{attribute 'Tc2GvlVarNames'}
VAR_GLOBAL
(*Master*)
(*Gerät 4 (CX5130-0121-M310), BOX 01*)
(*DP/DP-Kopppler*)
(*DP_State*)
(*
	R1_B01_PB_Zustand						AT %I*: USINT;
(*Daten*)
	R1_B01_StatusModule_I_Byte_1			AT %I*: USINT;
	R1_B01_StatusModule_I_Byte_2			AT %I*: USINT;
	R1_B01_StatusModule_I_Byte_5			AT %I*: USINT;
	R1_B01_StatusModule_I_Byte_6			AT %I*: USINT;
	R1_B01_ControlModule_O					AT %Q* :ARRAY [0..4] OF USINT;
	R1_B01_VolumeFlow_I						AT %I* :UDINT;
	R1_B01_PumpLiquidTemp_I					AT %I* :UDINT;
	R1_B01_OperationTime_I					AT %I* :UDINT;
	R1_B01_ActualSetpoint_I					AT %I* :UDINT;
	R1_B01_Frequency_I						AT %I* :UDINT;
	R1_B01_UserSetpoint_I					AT %I* :UDINT;
	R1_B01_DiffPressure_I					AT %I* :UDINT;
	R1_B01_RemoteTemp2						AT %I* :UDINT;
	R1_B01_HeatEnergyCounter_I				AT %I* :UDINT;
	R1_B01_HeatDiffTemp						AT %I* :UDINT;
	R1_B01_HeatPower						AT %I* :UDINT;  (* B0_SequenceNumber(1),B1AddressGenib(30),B2Class(11),B3Operation_Lenght(1),B4Data1(ID.34),Data(B5-B8) *)
	R1_B01_DirectDataReques_Temp_Geni		AT %Q* :PB_GenibusType;		(*ARRAY [0..8] OF USINT := 1, 255, 11, 1, 34, 0, 0, 0, 0;*)
	R1_B01_DirectDataReply_Temp_Geni		AT %I* :PB_GenibusType;		(*ARRAY [0..8] OF USINT;*)



	R1_B01_NumberOfStarts					AT %I*	: 	UDINT;
	R1_B01_ActualSetpoint					AT %I*	:	UDINT;
	R1_B01_OperationTime					AT %I*	: 	UDINT;
	R1_B01_Speed							AT %I*	:	UDINT;
	R1_B01_Energy							AT %I*	: 	UDINT;
	R1_B01_Power							AT %I*	:	UDINT;
	R1_B01_PowerElectronicsTemp				AT %I*	:	UDINT;
	R1_B01_FaultCode						AT %I*	:	USINT;
	R1_B01_Volume							AT %I*	:	UDINT;
	R1_B01_WarningCode						AT %I*	:	USINT;

(*Gerät 4 (CX5130-0121-M310), BOX 02*)
(*DP/DP-Kopppler*)
(*DP_State*)
	R1_B02_PB_Zustand						AT %I*: USINT;
(*Daten*)
	R1_B02_StatusModule_I_Byte_1			AT %I*: USINT;
	R1_B02_StatusModule_I_Byte_2			AT %I*: USINT;
	R1_B02_StatusModule_I_Byte_5			AT %I*: USINT;
	R1_B02_StatusModule_I_Byte_6			AT %I*: USINT;
	R1_B02_ControlModule_O					AT %Q* :ARRAY [0..4] OF USINT;
	R1_B02_VolumeFlow_I						AT %I* :UDINT;
	R1_B02_PumpLiquidTemp_I					AT %I* :UDINT;
	R1_B02_OperationTime_I					AT %I* :UDINT;
	R1_B02_ActualSetpoint_I					AT %I* :UDINT;
	R1_B02_Frequency_I						AT %I* :UDINT;
	R1_B02_UserSetpoint_I					AT %I* :UDINT;
	R1_B02_DiffPressure_I					AT %I* :UDINT;
	R1_B02_RemoteTemp2						AT %I* :UDINT;
	R1_B02_HeatEnergyCounter_I				AT %I* :UDINT;
	R1_B02_HeatDiffTemp						AT %I* :UDINT;
	R1_B02_HeatPower						AT %I* :UDINT;(* B0_SequenceNumber(1),B1AddressGenib(30),B2Class(11),B3Operation_Lenght(1),B4Data1(ID.34),Data(B5-B8) *)
	R1_B02_DirectDataReques_Temp_Geni		AT %Q* :PB_GenibusType;
	R1_B02_DirectDataReply_Temp_Geni		AT %I* :PB_GenibusType;


	R1_B02_NumberOfStarts					AT %I*	: 	UDINT;
	R1_B02_ActualSetpoint					AT %I*	:	UDINT;
	R1_B02_OperationTime					AT %I*	: 	UDINT;
	R1_B02_Speed							AT %I*	:	UDINT;
	R1_B02_Energy							AT %I*	: 	UDINT;
	R1_B02_Power							AT %I*	:	UDINT;
	R1_B02_PowerElectronicsTemp				AT %I*	:	UDINT;
	R1_B02_FaultCode						AT %I*	:	USINT;
	R1_B02_Volume							AT %I*	:	UDINT;
	R1_B02_WarningCode						AT %I*	:	USINT;

(*Gerät 4 (CX5130-0121-M310), BOX 03*)
(*DP/DP-Kopppler*)
(*DP_State*)
	R1_B03_PB_Zustand						AT %I*: USINT;
(*Daten*)
	R1_B03_StatusModule_I_Byte_1			AT %I*: USINT;
	R1_B03_StatusModule_I_Byte_2			AT %I*: USINT;
	R1_B03_StatusModule_I_Byte_5			AT %I*: USINT;
	R1_B03_StatusModule_I_Byte_6			AT %I*: USINT;
	R1_B03_ControlModule_O					AT %Q* :ARRAY [0..4] OF USINT;
	R1_B03_VolumeFlow_I						AT %I* :UDINT;
	R1_B03_PumpLiquidTemp_I					AT %I* :UDINT;
	R1_B03_OperationTime_I					AT %I* :UDINT;
	R1_B03_ActualSetpoint_I					AT %I* :UDINT;
	R1_B03_Frequency_I						AT %I* :UDINT;
	R1_B03_UserSetpoint_I					AT %I* :UDINT;
	R1_B03_DiffPressure_I					AT %I* :UDINT;
	R1_B03_RemoteTemp2						AT %I* :UDINT;
	R1_B03_HeatEnergyCounter_I				AT %I* :UDINT;
	R1_B03_HeatDiffTemp						AT %I* :UDINT;
	R1_B03_HeatPower						AT %I* :UDINT;(* B0_SequenceNumber(1),B1AddressGenib(30),B2Class(11),B3Operation_Lenght(1),B4Data1(ID.34),Data(B5-B8) *)
	R1_B03_DirectDataReques_Temp_Geni		AT %Q* :PB_GenibusType;
	R1_B03_DirectDataReply_Temp_Geni		AT %I* :PB_GenibusType;

	R1_B03_NumberOfStarts					AT %I*	: 	UDINT;
	R1_B03_ActualSetpoint					AT %I*	:	UDINT;
	R1_B03_OperationTime					AT %I*	: 	UDINT;
	R1_B03_Speed							AT %I*	:	UDINT;
	R1_B03_Energy							AT %I*	: 	UDINT;
	R1_B03_Power							AT %I*	:	UDINT;
	R1_B03_PowerElectronicsTemp				AT %I*	:	UDINT;
	R1_B03_FaultCode						AT %I*	:	USINT;
	R1_B03_Volume							AT %I*	:	UDINT;
	R1_B03_WarningCode						AT %I*	:	USINT;

(*Gerät 4 (CX5130-0121-M310), BOX 04*)
(*DP/DP-Kopppler*)
(*DP_State*)
	R1_B04_PB_Zustand						AT %I*: USINT;
(*Daten*)
	R1_B04_StatusModule_I_Byte_1			AT %I*: USINT;
	R1_B04_StatusModule_I_Byte_2			AT %I*: USINT;
	R1_B04_StatusModule_I_Byte_5			AT %I*: USINT;
	R1_B04_StatusModule_I_Byte_6			AT %I*: USINT;
	R1_B04_ControlModule_O					AT %Q* :ARRAY [0..4] OF USINT;
	R1_B04_VolumeFlow_I						AT %I* :UDINT;
	R1_B04_PumpLiquidTemp_I					AT %I* :UDINT;
	R1_B04_OperationTime_I					AT %I* :UDINT;
	R1_B04_ActualSetpoint_I					AT %I* :UDINT;
	R1_B04_Frequency_I						AT %I* :UDINT;
	R1_B04_UserSetpoint_I					AT %I* :UDINT;
	R1_B04_DiffPressure_I					AT %I* :UDINT;
	R1_B04_RemoteTemp2						AT %I* :UDINT;
	R1_B04_HeatEnergyCounter_I				AT %I* :UDINT;
	R1_B04_HeatDiffTemp						AT %I* :UDINT;
	R1_B04_HeatPower						AT %I* :UDINT;(* B0_SequenceNumber(1),B1AddressGenib(30),B2Class(11),B3Operation_Lenght(1),B4Data1(ID.34),Data(B5-B8) *)
	R1_B04_DirectDataReques_Temp_Geni		AT %Q* :PB_GenibusType;
	R1_B04_DirectDataReply_Temp_Geni		AT %I* :PB_GenibusType;


	R1_B04_NumberOfStarts					AT %I*	: 	UDINT;
	R1_B04_ActualSetpoint					AT %I*	:	UDINT;
	R1_B04_OperationTime					AT %I*	: 	UDINT;
	R1_B04_Speed							AT %I*	:	UDINT;
	R1_B04_Energy							AT %I*	: 	UDINT;
	R1_B04_Power							AT %I*	:	UDINT;
	R1_B04_PowerElectronicsTemp				AT %I*	:	UDINT;
	R1_B04_FaultCode						AT %I*	:	USINT;
	R1_B04_Volume							AT %I*	:	UDINT;
	R1_B04_WarningCode						AT %I*	:	USINT;


(*Gerät 4 (CX5130-0121-M310), BOX 05*)
(*DP/DP-Kopppler*)
(*DP_State*)
	R1_B05_PB_Zustand						AT %I*: USINT;
(*Daten*)
	R1_B05_StatusModule_I_Byte_1			AT %I*: USINT;
	R1_B05_StatusModule_I_Byte_2			AT %I*: USINT;
	R1_B05_StatusModule_I_Byte_5			AT %I*: USINT;
	R1_B05_StatusModule_I_Byte_6			AT %I*: USINT;
	R1_B05_ControlModule_O					AT %Q* :ARRAY [0..4] OF USINT;
	R1_B05_VolumeFlow_I						AT %I* :UDINT;
	R1_B05_PumpLiquidTemp_I					AT %I* :UDINT;
	R1_B05_OperationTime_I					AT %I* :UDINT;
	R1_B05_ActualSetpoint_I					AT %I* :UDINT;
	R1_B05_Frequency_I						AT %I* :UDINT;
	R1_B05_UserSetpoint_I					AT %I* :UDINT;
	R1_B05_DiffPressure_I					AT %I* :UDINT;
	R1_B05_RemoteTemp2						AT %I* :UDINT;
	R1_B05_HeatEnergyCounter_I				AT %I* :UDINT;
	R1_B05_HeatDiffTemp						AT %I* :UDINT;
	R1_B05_HeatPower						AT %I* :UDINT;(* B0_SequenceNumber(1),B1AddressGenib(30),B2Class(11),B3Operation_Lenght(1),B4Data1(ID.34),Data(B5-B8) *)
	R1_B05_DirectDataReques_Temp_Geni		AT %Q* :PB_GenibusType;
	R1_B05_DirectDataReply_Temp_Geni		AT %I* :PB_GenibusType;

	R1_B05_NumberOfStarts					AT %I*	: 	UDINT;
	R1_B05_ActualSetpoint					AT %I*	:	UDINT;
	R1_B05_OperationTime					AT %I*	: 	UDINT;
	R1_B05_Speed							AT %I*	:	UDINT;
	R1_B05_Energy							AT %I*	: 	UDINT;
	R1_B05_Power							AT %I*	:	UDINT;
	R1_B05_PowerElectronicsTemp				AT %I*	:	UDINT;
	R1_B05_FaultCode						AT %I*	:	USINT;
	R1_B05_Volume							AT %I*	:	UDINT;
	R1_B05_WarningCode						AT %I*	:	USINT;


(*Gerät 4 (CX5130-0121-M310), BOX 06*)
(*DP/DP-Kopppler*)
(*DP_State*)
	R1_B06_PB_Zustand						AT %I*: USINT;
(*Daten*)
	R1_B06_StatusModule_I_Byte_1			AT %I*: USINT;
	R1_B06_StatusModule_I_Byte_2			AT %I*: USINT;
	R1_B06_StatusModule_I_Byte_5			AT %I*: USINT;
	R1_B06_StatusModule_I_Byte_6			AT %I*: USINT;
	R1_B06_ControlModule_O					AT %Q* :ARRAY [0..4] OF USINT;
	R1_B06_VolumeFlow_I						AT %I* :UDINT;
	R1_B06_PumpLiquidTemp_I					AT %I* :UDINT;
	R1_B06_OperationTime_I					AT %I* :UDINT;
	R1_B06_ActualSetpoint_I					AT %I* :UDINT;
	R1_B06_Frequency_I						AT %I* :UDINT;
	R1_B06_UserSetpoint_I					AT %I* :UDINT;
	R1_B06_DiffPressure_I					AT %I* :UDINT;
	R1_B06_RemoteTemp2						AT %I* :UDINT;
	R1_B06_HeatEnergyCounter_I				AT %I* :UDINT;
	R1_B06_HeatDiffTemp						AT %I* :UDINT;
	R1_B06_HeatPower						AT %I* :UDINT;(* B0_SequenceNumber(1),B1AddressGenib(30),B2Class(11),B3Operation_Lenght(1),B4Data1(ID.34),Data(B5-B8) *)
	R1_B06_DirectDataReques_Temp_Geni		AT %Q* :PB_GenibusType;
	R1_B06_DirectDataReply_Temp_Geni		AT %I* :PB_GenibusType;

	R1_B06_NumberOfStarts					AT %I*	: 	UDINT;
	R1_B06_ActualSetpoint					AT %I*	:	UDINT;
	R1_B06_OperationTime					AT %I*	: 	UDINT;
	R1_B06_Speed							AT %I*	:	UDINT;
	R1_B06_Energy							AT %I*	: 	UDINT;
	R1_B06_Power							AT %I*	:	UDINT;
	R1_B06_PowerElectronicsTemp				AT %I*	:	UDINT;
	R1_B06_FaultCode						AT %I*	:	USINT;
	R1_B06_Volume							AT %I*	:	UDINT;
	R1_B06_WarningCode						AT %I*	:	USINT;

(*Gerät 4 (CX5130-0121-M310), BOX 07*)                           (*Pumpe entfallen*)
(*DP/DP-Kopppler*)
(*DP_State*)
	R1_B07_PB_Zustand						AT %I*: USINT;
(*Daten*)
	R1_B07_StatusModule_I_Byte_1			AT %I*: USINT;
	R1_B07_StatusModule_I_Byte_2			AT %I*: USINT;
	R1_B07_StatusModule_I_Byte_5			AT %I*: USINT;
	R1_B07_StatusModule_I_Byte_6			AT %I*: USINT;
	R1_B07_ControlModule_O					AT %Q* :ARRAY [0..4] OF USINT;
	R1_B07_VolumeFlow_I						AT %I* :UDINT;
	R1_B07_PumpLiquidTemp_I					AT %I* :UDINT;
	R1_B07_OperationTime_I					AT %I* :UDINT;
	R1_B07_ActualSetpoint_I					AT %I* :UDINT;
	R1_B07_Frequency_I						AT %I* :UDINT;
	R1_B07_UserSetpoint_I					AT %I* :UDINT;
	R1_B07_DiffPressure_I					AT %I* :UDINT;
	R1_B07_RemoteTemp2						AT %I* :UDINT;
	R1_B07_HeatEnergyCounter_I				AT %I* :UDINT;
	R1_B07_HeatDiffTemp						AT %I* :UDINT;
	R1_B07_HeatPower						AT %I* :UDINT;

	R1_B07_NumberOfStarts					AT %I*	: 	UDINT;
	R1_B07_ActualSetpoint					AT %I*	:	UDINT;
	R1_B07_OperationTime					AT %I*	: 	UDINT;
	R1_B07_Speed							AT %I*	:	UDINT;
	R1_B07_Energy							AT %I*	: 	UDINT;
	R1_B07_Power							AT %I*	:	UDINT;
	R1_B07_PowerElectronicsTemp				AT %I*	:	UDINT;
	R1_B07_FaultCode						AT %I*	:	USINT;
	R1_B07_Volume							AT %I*	:	UDINT;
	R1_B07_WarningCode						AT %I*	:	USINT;


(*Gerät 4 (CX5130-0121-M310), BOX 08*)							  (*Pumpe entfallen*)
(*DP/DP-Kopppler*)
(*DP_State*)
	R1_B08_PB_Zustand						AT %I*: USINT;
(*Daten*)
	R1_B08_StatusModule_I_Byte_1			AT %I*: USINT;
	R1_B08_StatusModule_I_Byte_2			AT %I*: USINT;
	R1_B08_StatusModule_I_Byte_5			AT %I*: USINT;
	R1_B08_StatusModule_I_Byte_6			AT %I*: USINT;
	R1_B08_ControlModule_O					AT %Q* :ARRAY [0..4] OF USINT;
	R1_B08_VolumeFlow_I						AT %I* :UDINT;
	R1_B08_PumpLiquidTemp_I					AT %I* :UDINT;
	R1_B08_OperationTime_I					AT %I* :UDINT;
	R1_B08_ActualSetpoint_I					AT %I* :UDINT;
	R1_B08_Frequency_I						AT %I* :UDINT;
	R1_B08_UserSetpoint_I					AT %I* :UDINT;
	R1_B08_DiffPressure_I					AT %I* :UDINT;
	R1_B08_RemoteTemp2						AT %I* :UDINT;
	R1_B08_HeatEnergyCounter_I				AT %I* :UDINT;
	R1_B08_HeatDiffTemp						AT %I* :UDINT;
	R1_B08_HeatPower						AT %I* :UDINT;

	R1_B08_NumberOfStarts					AT %I*	: 	UDINT;
	R1_B08_ActualSetpoint					AT %I*	:	UDINT;
	R1_B08_OperationTime					AT %I*	: 	UDINT;
	R1_B08_Speed							AT %I*	:	UDINT;
	R1_B08_Energy							AT %I*	: 	UDINT;
	R1_B08_Power							AT %I*	:	UDINT;
	R1_B08_PowerElectronicsTemp				AT %I*	:	UDINT;
	R1_B08_FaultCode						AT %I*	:	USINT;
	R1_B08_Volume							AT %I*	:	UDINT;
	R1_B08_WarningCode						AT %I*	:	USINT;

(*Gerät 4 (CX5130-0121-M310), BOX 09*)
(*DP/DP-Kopppler*)
(*DP_State*)
	R1_B09_PB_Zustand						AT %I*: USINT;
(*Daten*)
	R1_B09_StatusModule_I_Byte_1			AT %I*: USINT;
	R1_B09_StatusModule_I_Byte_2			AT %I*: USINT;
	R1_B09_StatusModule_I_Byte_5			AT %I*: USINT;
	R1_B09_StatusModule_I_Byte_6			AT %I*: USINT;
	R1_B09_ControlModule_O					AT %Q* :ARRAY [0..4] OF USINT;
	R1_B09_VolumeFlow_I						AT %I* :UDINT;
	R1_B09_PumpLiquidTemp_I					AT %I* :UDINT;
	R1_B09_OperationTime_I					AT %I* :UDINT;
	R1_B09_ActualSetpoint_I					AT %I* :UDINT;
	R1_B09_Frequency_I						AT %I* :UDINT;
	R1_B09_UserSetpoint_I					AT %I* :UDINT;
	R1_B09_DiffPressure_I					AT %I* :UDINT;
	R1_B09_RemoteTemp2						AT %I* :UDINT;
	R1_B09_HeatEnergyCounter_I				AT %I* :UDINT;
	R1_B09_HeatDiffTemp						AT %I* :UDINT;
	R1_B09_HeatPower						AT %I* :UDINT;(* B0_SequenceNumber(1),B1AddressGenib(30),B2Class(11),B3Operation_Lenght(1),B4Data1(ID.34),Data(B5-B8) *)
	R1_B09_DirectDataReques_Temp_Geni		AT %Q* :PB_GenibusType;
	R1_B09_DirectDataReply_Temp_Geni		AT %I* :PB_GenibusType;

	R1_B09_NumberOfStarts					AT %I*	: 	UDINT;
	R1_B09_ActualSetpoint					AT %I*	:	UDINT;
	R1_B09_OperationTime					AT %I*	: 	UDINT;
	R1_B09_Speed							AT %I*	:	UDINT;
	R1_B09_Energy							AT %I*	: 	UDINT;
	R1_B09_Power							AT %I*	:	UDINT;
	R1_B09_PowerElectronicsTemp				AT %I*	:	UDINT;
	R1_B09_FaultCode						AT %I*	:	USINT;
	R1_B09_Volume							AT %I*	:	UDINT;
	R1_B09_WarningCode						AT %I*	:	USINT;

(*Gerät 4 (CX5130-0121-M310), BOX 10*)
(*DP/DP-Kopppler*)
(*DP_State*)
	R1_B10_PB_Zustand						AT %I*: USINT;
(*Daten*)
	R1_B10_StatusModule_I_Byte_1			AT %I*: USINT;
	R1_B10_StatusModule_I_Byte_2			AT %I*: USINT;
	R1_B10_StatusModule_I_Byte_5			AT %I*: USINT;
	R1_B10_StatusModule_I_Byte_6			AT %I*: USINT;
	R1_B10_ControlModule_O					AT %Q* :ARRAY [0..4] OF USINT;
	R1_B10_VolumeFlow_I						AT %I* :UDINT;
	R1_B10_PumpLiquidTemp_I					AT %I* :UDINT;
	R1_B10_OperationTime_I					AT %I* :UDINT;
	R1_B10_ActualSetpoint_I					AT %I* :UDINT;
	R1_B10_Frequency_I						AT %I* :UDINT;
	R1_B10_UserSetpoint_I					AT %I* :UDINT;
	R1_B10_DiffPressure_I					AT %I* :UDINT;
	R1_B10_RemoteTemp2						AT %I* :UDINT;
	R1_B10_HeatEnergyCounter_I				AT %I* :UDINT;
	R1_B10_HeatDiffTemp						AT %I* :UDINT;
	R1_B10_HeatPower						AT %I* :UDINT;(* B0_SequenceNumber(1),B1AddressGenib(30),B2Class(11),B3Operation_Lenght(1),B4Data1(ID.34),Data(B5-B8) *)
	R1_B10_DirectDataReques_Temp_Geni		AT %Q* :PB_GenibusType;
	R1_B10_DirectDataReply_Temp_Geni		AT %I* :PB_GenibusType;

	R1_B10_NumberOfStarts					AT %I*	: 	UDINT;
	R1_B10_ActualSetpoint					AT %I*	:	UDINT;
	R1_B10_OperationTime					AT %I*	: 	UDINT;
	R1_B10_Speed							AT %I*	:	UDINT;
	R1_B10_Energy							AT %I*	: 	UDINT;
	R1_B10_Power							AT %I*	:	UDINT;
	R1_B10_PowerElectronicsTemp				AT %I*	:	UDINT;
	R1_B10_FaultCode						AT %I*	:	USINT;
	R1_B10_Volume							AT %I*	:	UDINT;
	R1_B10_WarningCode						AT %I*	:	USINT;

(*Gerät 4 (CX5130-0121-M310), BOX 11*)
(*DP/DP-Kopppler*)
(*DP_State*)
	R1_B11_PB_Zustand						AT %I*: USINT;
(*Daten*)
	R1_B11_StatusModule_I_Byte_1			AT %I*: USINT;
	R1_B11_StatusModule_I_Byte_2			AT %I*: USINT;
	R1_B11_StatusModule_I_Byte_5			AT %I*: USINT;
	R1_B11_StatusModule_I_Byte_6			AT %I*: USINT;
	R1_B11_ControlModule_O					AT %Q* :ARRAY [0..4] OF USINT;
	R1_B11_VolumeFlow_I						AT %I* :UDINT;
	R1_B11_PumpLiquidTemp_I					AT %I* :UDINT;
	R1_B11_OperationTime_I					AT %I* :UDINT;
	R1_B11_ActualSetpoint_I					AT %I* :UDINT;
	R1_B11_Frequency_I						AT %I* :UDINT;
	R1_B11_UserSetpoint_I					AT %I* :UDINT;
	R1_B11_DiffPressure_I					AT %I* :UDINT;
	R1_B11_RemoteTemp2						AT %I* :UDINT;
	R1_B11_HeatEnergyCounter_I				AT %I* :UDINT;
	R1_B11_HeatDiffTemp						AT %I* :UDINT;
	R1_B11_HeatPower						AT %I* :UDINT;(* B0_SequenceNumber(1),B1AddressGenib(30),B2Class(11),B3Operation_Lenght(1),B4Data1(ID.34),Data(B5-B8) *)
	R1_B11_DirectDataReques_Temp_Geni		AT %Q* :PB_GenibusType;
	R1_B11_DirectDataReply_Temp_Geni		AT %I* :PB_GenibusType;


	R1_B11_NumberOfStarts					AT %I*	: 	UDINT;
	R1_B11_ActualSetpoint					AT %I*	:	UDINT;
	R1_B11_OperationTime					AT %I*	: 	UDINT;
	R1_B11_Speed							AT %I*	:	UDINT;
	R1_B11_Energy							AT %I*	: 	UDINT;
	R1_B11_Power							AT %I*	:	UDINT;
	R1_B11_PowerElectronicsTemp				AT %I*	:	UDINT;
	R1_B11_FaultCode						AT %I*	:	USINT;
	R1_B11_Volume							AT %I*	:	UDINT;
	R1_B11_WarningCode						AT %I*	:	USINT;

(*Gerät 4 (CX5130-0121-M310), BOX 12*)								  (*Pumpe entfallen*)
(*DP/DP-Kopppler*)
(*DP_State*)
	R1_B12_PB_Zustand						AT %I*: USINT;
(*Daten*)
	R1_B12_StatusModule_I_Byte_1			AT %I*: USINT;
	R1_B12_StatusModule_I_Byte_2			AT %I*: USINT;
	R1_B12_StatusModule_I_Byte_5			AT %I*: USINT;
	R1_B12_StatusModule_I_Byte_6			AT %I*: USINT;
	R1_B12_ControlModule_O					AT %Q* :ARRAY [0..4] OF USINT;
	R1_B12_VolumeFlow_I						AT %I* :UDINT;
	R1_B12_PumpLiquidTemp_I					AT %I* :UDINT;
	R1_B12_OperationTime_I					AT %I* :UDINT;
	R1_B12_ActualSetpoint_I					AT %I* :UDINT;
	R1_B12_Frequency_I						AT %I* :UDINT;
	R1_B12_UserSetpoint_I					AT %I* :UDINT;
	R1_B12_DiffPressure_I					AT %I* :UDINT;
	R1_B12_RemoteTemp2						AT %I* :UDINT;
	R1_B12_HeatEnergyCounter_I				AT %I* :UDINT;
	R1_B12_HeatDiffTemp						AT %I* :UDINT;
	R1_B12_HeatPower						AT %I* :UDINT;

(*Gerät 4 (CX5130-0121-M310), BOX 13*)
(*DP/DP-Kopppler*)
(*DP_State*)
	R1_B13_PB_Zustand						AT %I*: USINT;
(*Daten*)
	R1_B13_StatusModule_I_Byte_1			AT %I*: USINT;
	R1_B13_StatusModule_I_Byte_2			AT %I*: USINT;
	R1_B13_StatusModule_I_Byte_5			AT %I*: USINT;
	R1_B13_StatusModule_I_Byte_6			AT %I*: USINT;
	R1_B13_ControlModule_O					AT %Q* :ARRAY [0..4] OF USINT;
	R1_B13_VolumeFlow_I						AT %I* :UDINT;
	R1_B13_PumpLiquidTemp_I					AT %I* :UDINT;
	R1_B13_OperationTime_I					AT %I* :UDINT;
	R1_B13_ActualSetpoint_I					AT %I* :UDINT;
	R1_B13_Frequency_I						AT %I* :UDINT;
	R1_B13_UserSetpoint_I					AT %I* :UDINT;
	R1_B13_DiffPressure_I					AT %I* :UDINT;
	R1_B13_RemoteTemp2						AT %I* :UDINT;
	R1_B13_HeatEnergyCounter_I				AT %I* :UDINT;
	R1_B13_HeatDiffTemp						AT %I* :UDINT;
	R1_B13_HeatPower						AT %I* :UDINT;(* B0_SequenceNumber(1),B1AddressGenib(30),B2Class(11),B3Operation_Lenght(1),B4Data1(ID.34),Data(B5-B8) *)
	R1_B13_DirectDataReques_Temp_Geni		AT %Q* :PB_GenibusType;
	R1_B13_DirectDataReply_Temp_Geni		AT %I* :PB_GenibusType;


	R1_B13_NumberOfStarts					AT %I*	: 	UDINT;
	R1_B13_ActualSetpoint					AT %I*	:	UDINT;
	R1_B13_OperationTime					AT %I*	: 	UDINT;
	R1_B13_Speed							AT %I*	:	UDINT;
	R1_B13_Energy							AT %I*	: 	UDINT;
	R1_B13_Power							AT %I*	:	UDINT;
	R1_B13_PowerElectronicsTemp				AT %I*	:	UDINT;
	R1_B13_FaultCode						AT %I*	:	USINT;
	R1_B13_Volume							AT %I*	:	UDINT;
	R1_B13_WarningCode						AT %I*	:	USINT;

(*Gerät 4 (CX5130-0121-M310), BOX 14*)
(*DP/DP-Kopppler*)
(*DP_State*)
	R1_B14_PB_Zustand						AT %I*: USINT;
(*Daten*)
	R1_B14_StatusModule_I_Byte_1			AT %I*: USINT;
	R1_B14_StatusModule_I_Byte_2			AT %I*: USINT;
	R1_B14_StatusModule_I_Byte_5			AT %I*: USINT;
	R1_B14_StatusModule_I_Byte_6			AT %I*: USINT;
	R1_B14_ControlModule_O					AT %Q* :ARRAY [0..4] OF USINT;
	R1_B14_VolumeFlow_I						AT %I* :UDINT;
	R1_B14_PumpLiquidTemp_I					AT %I* :UDINT;
	R1_B14_OperationTime_I					AT %I* :UDINT;
	R1_B14_ActualSetpoint_I					AT %I* :UDINT;
	R1_B14_Frequency_I						AT %I* :UDINT;
	R1_B14_UserSetpoint_I					AT %I* :UDINT;
	R1_B14_DiffPressure_I					AT %I* :UDINT;
	R1_B14_RemoteTemp2						AT %I* :UDINT;
	R1_B14_HeatEnergyCounter_I				AT %I* :UDINT;
	R1_B14_HeatDiffTemp						AT %I* :UDINT;
	R1_B14_HeatPower						AT %I* :UDINT;(* B0_SequenceNumber(1),B1AddressGenib(30),B2Class(11),B3Operation_Lenght(1),B4Data1(ID.34),Data(B5-B8) *)
	R1_B14_DirectDataReques_Temp_Geni		AT %Q* :PB_GenibusType;
	R1_B14_DirectDataReply_Temp_Geni		AT %I* :PB_GenibusType;


	R1_B14_NumberOfStarts					AT %I*	: 	UDINT;
	R1_B14_ActualSetpoint					AT %I*	:	UDINT;
	R1_B14_OperationTime					AT %I*	: 	UDINT;
	R1_B14_Speed							AT %I*	:	UDINT;
	R1_B14_Energy							AT %I*	: 	UDINT;
	R1_B14_Power							AT %I*	:	UDINT;
	R1_B14_PowerElectronicsTemp				AT %I*	:	UDINT;
	R1_B14_FaultCode						AT %I*	:	USINT;
	R1_B14_Volume							AT %I*	:	UDINT;
	R1_B14_WarningCode						AT %I*	:	USINT;

(*Gerät 4 (CX5130-0121-M310), BOX 15*)
(*DP/DP-Kopppler*)
(*DP_State*)
	R1_B15_PB_Zustand						AT %I*: USINT;
(*Daten*)
	R1_B15_StatusModule_I_Byte_1			AT %I*: USINT;
	R1_B15_StatusModule_I_Byte_2			AT %I*: USINT;
	R1_B15_StatusModule_I_Byte_5			AT %I*: USINT;
	R1_B15_StatusModule_I_Byte_6			AT %I*: USINT;
	R1_B15_ControlModule_O					AT %Q* :ARRAY [0..4] OF USINT;
	R1_B15_VolumeFlow_I						AT %I* :UDINT;
	R1_B15_PumpLiquidTemp_I					AT %I* :UDINT;
	R1_B15_OperationTime_I					AT %I* :UDINT;
	R1_B15_ActualSetpoint_I					AT %I* :UDINT;
	R1_B15_Frequency_I						AT %I* :UDINT;
	R1_B15_UserSetpoint_I					AT %I* :UDINT;
	R1_B15_DiffPressure_I					AT %I* :UDINT;
	R1_B15_RemoteTemp2						AT %I* :UDINT;
	R1_B15_HeatEnergyCounter_I				AT %I* :UDINT;
	R1_B15_HeatDiffTemp						AT %I* :UDINT;
	R1_B15_HeatPower						AT %I* :UDINT;(* B0_SequenceNumber(1),B1AddressGenib(30),B2Class(11),B3Operation_Lenght(1),B4Data1(ID.34),Data(B5-B8) *)
	R1_B15_DirectDataReques_Temp_Geni		AT %Q* :PB_GenibusType;
	R1_B15_DirectDataReply_Temp_Geni		AT %I* :PB_GenibusType;


	R1_B15_NumberOfStarts					AT %I*	: 	UDINT;
	R1_B15_ActualSetpoint					AT %I*	:	UDINT;
	R1_B15_OperationTime					AT %I*	: 	UDINT;
	R1_B15_Speed							AT %I*	:	UDINT;
	R1_B15_Energy							AT %I*	: 	UDINT;
	R1_B15_Power							AT %I*	:	UDINT;
	R1_B15_PowerElectronicsTemp				AT %I*	:	UDINT;
	R1_B15_FaultCode						AT %I*	:	USINT;
	R1_B15_Volume							AT %I*	:	UDINT;
	R1_B15_WarningCode						AT %I*	:	USINT;

(*Gerät 4 (CX5130-0121-M310), BOX 16*)
(*DP/DP-Kopppler*)
(*DP_State*)
	R1_B16_PB_Zustand						AT %I*: USINT;
(*Daten*)
	R1_B16_StatusModule_I_Byte_1			AT %I*: USINT;
	R1_B16_StatusModule_I_Byte_2			AT %I*: USINT;
	R1_B16_StatusModule_I_Byte_5			AT %I*: USINT;
	R1_B16_StatusModule_I_Byte_6			AT %I*: USINT;
	R1_B16_ControlModule_O					AT %Q* :ARRAY [0..4] OF USINT;
	R1_B16_VolumeFlow_I						AT %I* :UDINT;
	R1_B16_PumpLiquidTemp_I					AT %I* :UDINT;
	R1_B16_OperationTime_I					AT %I* :UDINT;
	R1_B16_ActualSetpoint_I					AT %I* :UDINT;
	R1_B16_Frequency_I						AT %I* :UDINT;
	R1_B16_UserSetpoint_I					AT %I* :UDINT;
	R1_B16_DiffPressure_I					AT %I* :UDINT;
	R1_B16_RemoteTemp2						AT %I* :UDINT;
	R1_B16_HeatEnergyCounter_I				AT %I* :UDINT;
	R1_B16_HeatDiffTemp						AT %I* :UDINT;
	R1_B16_HeatPower						AT %I* :UDINT;(* B0_SequenceNumber(1),B1AddressGenib(30),B2Class(11),B3Operation_Lenght(1),B4Data1(ID.34),Data(B5-B8) *)
	R1_B16_DirectDataReques_Temp_Geni		AT %Q* :PB_GenibusType;
	R1_B16_DirectDataReply_Temp_Geni		AT %I* :PB_GenibusType;


	R1_B16_NumberOfStarts					AT %I*	: 	UDINT;
	R1_B16_ActualSetpoint					AT %I*	:	UDINT;
	R1_B16_OperationTime					AT %I*	: 	UDINT;
	R1_B16_Speed							AT %I*	:	UDINT;
	R1_B16_Energy							AT %I*	: 	UDINT;
	R1_B16_Power							AT %I*	:	UDINT;
	R1_B16_PowerElectronicsTemp				AT %I*	:	UDINT;
	R1_B16_FaultCode						AT %I*	:	USINT;
	R1_B16_Volume							AT %I*	:	UDINT;
	R1_B16_WarningCode						AT %I*	:	USINT;

(*Gerät 4 (CX5130-0121-M310), BOX 17*)
(*DP/DP-Kopppler*)
(*DP_State*)
	R1_B17_PB_Zustand						AT %I*: USINT;
(*Daten*)
	R1_B17_StatusModule_I_Byte_1			AT %I*: USINT;
	R1_B17_StatusModule_I_Byte_2			AT %I*: USINT;
	R1_B17_StatusModule_I_Byte_5			AT %I*: USINT;
	R1_B17_StatusModule_I_Byte_6			AT %I*: USINT;
	R1_B17_ControlModule_O					AT %Q* :ARRAY [0..4] OF USINT;
	R1_B17_VolumeFlow_I						AT %I* :UDINT;
	R1_B17_PumpLiquidTemp_I					AT %I* :UDINT;
	R1_B17_OperationTime_I					AT %I* :UDINT;
	R1_B17_ActualSetpoint_I					AT %I* :UDINT;
	R1_B17_Frequency_I						AT %I* :UDINT;
	R1_B17_UserSetpoint_I					AT %I* :UDINT;
	R1_B17_DiffPressure_I					AT %I* :UDINT;
	R1_B17_RemoteTemp2						AT %I* :UDINT;
	R1_B17_HeatEnergyCounter_I				AT %I* :UDINT;
	R1_B17_HeatDiffTemp						AT %I* :UDINT;
	R1_B17_HeatPower						AT %I* :UDINT;(* B0_SequenceNumber(1),B1AddressGenib(30),B2Class(11),B3Operation_Lenght(1),B4Data1(ID.34),Data(B5-B8) *)
	R1_B17_DirectDataReques_Temp_Geni		AT %Q* :PB_GenibusType;
	R1_B17_DirectDataReply_Temp_Geni		AT %I* :PB_GenibusType;


	R1_B17_NumberOfStarts					AT %I*	: 	UDINT;
	R1_B17_ActualSetpoint					AT %I*	:	UDINT;
	R1_B17_OperationTime					AT %I*	: 	UDINT;
	R1_B17_Speed							AT %I*	:	UDINT;
	R1_B17_Energy							AT %I*	: 	UDINT;
	R1_B17_Power							AT %I*	:	UDINT;
	R1_B17_PowerElectronicsTemp				AT %I*	:	UDINT;
	R1_B17_FaultCode						AT %I*	:	USINT;
	R1_B17_Volume							AT %I*	:	UDINT;
	R1_B17_WarningCode						AT %I*	:	USINT;

(*Gerät 4 (CX5130-0121-M310), BOX 18*)
(*DP/DP-Kopppler*)
		(* Variablen in Globale Variablen   AC_PB_Var definiert
		Anbindung Atlas Copco MK5 Profibus Gateway Compressor *)


(* Janitza UMG 604 in Druckluftkompressor*)
	R1_B19_Request							AT %Q* 	:	BYTE;
	R1_B19_In								AT %I*	:	ARRAY[0..31] OF UINT;


(*Master*)
(*Gerät 6 (EL6731), BOX 01*)
(*DP/DP-Kopppler*)
(*DP_State*)
	R2_B01_PB_Zustand						AT %I*: USINT;
(*Daten*)
	R2_B01_StatusModule_I_Byte_1			AT %I*: USINT;
	R2_B01_StatusModule_I_Byte_2			AT %I*: USINT;
	R2_B01_StatusModule_I_Byte_5			AT %I*: USINT;
	R2_B01_StatusModule_I_Byte_6			AT %I*: USINT;
	R2_B01_ControlModule_O					AT %Q* :ARRAY [0..4] OF USINT;  (*Control Modul muss getestet werden*)
	R2_B01_VolumeFlow_I						AT %I* :UDINT;
	R2_B01_PumpLiquidTemp_I					AT %I* :UDINT;
	R2_B01_OperationTime_I					AT %I* :UDINT;
	R2_B01_ActualSetpoint_I					AT %I* :UDINT;
	R2_B01_Frequency_I						AT %I* :UDINT;
	R2_B01_UserSetpoint_I					AT %I* :UDINT;
	R2_B01_DiffPressure_I					AT %I* :UDINT;
	R2_B01_RemoteTemp2						AT %I* :UDINT;
	R2_B01_HeatEnergyCounter_I				AT %I* :UDINT;
	R2_B01_HeatDiffTemp						AT %I* :UDINT;
	R2_B01_HeatPower						AT %I* :UDINT;(* B0_SequenceNumber(1),B1AddressGenib(30),B2Class(11),B3Operation_Lenght(1),B4Data1(ID.34),Data(B5-B8) *)
	R2_B01_DirectDataReques_Temp_Geni		AT %Q* :PB_GenibusType;
	R2_B01_DirectDataReply_Temp_Geni		AT %I* :PB_GenibusType;

	R2_B01_NumberOfStarts					AT %I*	: 	UDINT;
	R2_B01_ActualSetpoint					AT %I*	:	UDINT;
	R2_B01_OperationTime					AT %I*	: 	UDINT;
	R2_B01_Speed							AT %I*	:	UDINT;
	R2_B01_Energy							AT %I*	: 	UDINT;
	R2_B01_Power							AT %I*	:	UDINT;
	R2_B01_PowerElectronicsTemp				AT %I*	:	UDINT;
	R2_B01_FaultCode						AT %I*	:	USINT;
	R2_B01_Volume							AT %I*	:	UDINT;
	R2_B01_WarningCode						AT %I*	:	USINT;


(*Gerät 6 (EL6731), BOX 02*)
(*DP/DP-Kopppler*)
(*DP_State*)
	R2_B02_PB_Zustand						AT %I*: USINT;
(*Daten*)
	R2_B02_StatusModule_I_Byte_1			AT %I*: USINT;
	R2_B02_StatusModule_I_Byte_2			AT %I*: USINT;
	R2_B02_StatusModule_I_Byte_5			AT %I*: USINT;
	R2_B02_StatusModule_I_Byte_6			AT %I*: USINT;
	R2_B02_ControlModule_O					AT %Q* :ARRAY [0..4] OF USINT;
	R2_B02_VolumeFlow_I						AT %I* :UDINT;
	R2_B02_PumpLiquidTemp_I					AT %I* :UDINT;
	R2_B02_OperationTime_I					AT %I* :UDINT;
	R2_B02_ActualSetpoint_I					AT %I* :UDINT;
	R2_B02_Frequency_I						AT %I* :UDINT;
	R2_B02_UserSetpoint_I					AT %I* :UDINT;
	R2_B02_DiffPressure_I					AT %I* :UDINT;
	R2_B02_RemoteTemp2						AT %I* :UDINT;
	R2_B02_HeatEnergyCounter_I				AT %I* :UDINT;
	R2_B02_HeatDiffTemp						AT %I* :UDINT;
	R2_B02_HeatPower						AT %I* :UDINT;(* B0_SequenceNumber(1),B1AddressGenib(30),B2Class(11),B3Operation_Lenght(1),B4Data1(ID.34),Data(B5-B8) *)
	R2_B02_DirectDataReques_Temp_Geni		AT %Q* :PB_GenibusType;
	R2_B02_DirectDataReply_Temp_Geni		AT %I* :PB_GenibusType;

	R2_B02_NumberOfStarts					AT %I*	: 	UDINT;
	R2_B02_ActualSetpoint					AT %I*	:	UDINT;
	R2_B02_OperationTime					AT %I*	: 	UDINT;
	R2_B02_Speed							AT %I*	:	UDINT;
	R2_B02_Energy							AT %I*	: 	UDINT;
	R2_B02_Power							AT %I*	:	UDINT;
	R2_B02_PowerElectronicsTemp				AT %I*	:	UDINT;
	R2_B02_FaultCode						AT %I*	:	USINT;
	R2_B02_Volume							AT %I*	:	UDINT;
	R2_B02_WarningCode						AT %I*	:	USINT;


(*Gerät 6 (EL6731), BOX 03*)
(*DP/DP-Kopppler*)
(*DP_State*)
	R2_B03_PB_Zustand						AT %I*: USINT;
(*Daten*)
	R2_B03_StatusModule_I_Byte_1			AT %I*: USINT;
	R2_B03_StatusModule_I_Byte_2			AT %I*: USINT;
	R2_B03_StatusModule_I_Byte_5			AT %I*: USINT;
	R2_B03_StatusModule_I_Byte_6			AT %I*: USINT;
	R2_B03_ControlModule_O					AT %Q* :ARRAY [0..4] OF USINT;
	R2_B03_VolumeFlow_I						AT %I* :UDINT;
	R2_B03_PumpLiquidTemp_I					AT %I* :UDINT;
	R2_B03_OperationTime_I					AT %I* :UDINT;
	R2_B03_ActualSetpoint_I					AT %I* :UDINT;
	R2_B03_Frequency_I						AT %I* :UDINT;
	R2_B03_UserSetpoint_I					AT %I* :UDINT;
	R2_B03_DiffPressure_I					AT %I* :UDINT;
	R2_B03_RemoteTemp2						AT %I* :UDINT;
	R2_B03_HeatEnergyCounter_I				AT %I* :UDINT;
	R2_B03_HeatDiffTemp						AT %I* :UDINT;
	R2_B03_HeatPower						AT %I* :UDINT;(* B0_SequenceNumber(1),B1AddressGenib(30),B2Class(11),B3Operation_Lenght(1),B4Data1(ID.34),Data(B5-B8) *)
	R2_B03_DirectDataReques_Temp_Geni		AT %Q* :PB_GenibusType;
	R2_B03_DirectDataReply_Temp_Geni		AT %I* :PB_GenibusType;

	R2_B03_NumberOfStarts					AT %I*	: 	UDINT;
	R2_B03_ActualSetpoint					AT %I*	:	UDINT;
	R2_B03_OperationTime					AT %I*	: 	UDINT;
	R2_B03_Speed							AT %I*	:	UDINT;
	R2_B03_Energy							AT %I*	: 	UDINT;
	R2_B03_Power							AT %I*	:	UDINT;
	R2_B03_PowerElectronicsTemp				AT %I*	:	UDINT;
	R2_B03_FaultCode						AT %I*	:	USINT;
	R2_B03_Volume							AT %I*	:	UDINT;
	R2_B03_WarningCode						AT %I*	:	USINT;


(*Gerät 6 (EL6731), BOX 04*)
(*DP/DP-Kopppler*)
(*DP_State*)
	R2_B04_PB_Zustand						AT %I*: USINT;
(*Daten*)
	R2_B04_StatusModule_I_Byte_1			AT %I*: USINT;
	R2_B04_StatusModule_I_Byte_2			AT %I*: USINT;
	R2_B04_StatusModule_I_Byte_5			AT %I*: USINT;
	R2_B04_StatusModule_I_Byte_6				AT %I*	:	 USINT;
	R2_B04_ControlModule_O					AT %Q* 	:	ARRAY [0..4] OF USINT;
	R2_B04_VolumeFlow_I						AT %I* 	:	UDINT;
	R2_B04_PumpLiquidTemp_I				AT %I* 	:	UDINT;
	R2_B04_OperationTime_I					AT %I* 	:	UDINT;
	R2_B04_ActualSetpoint_I					AT %I* 	:	UDINT;
	R2_B04_Frequency_I						AT %I* 	:	UDINT;
	R2_B04_UserSetpoint_I					AT %I* 	:	UDINT;
	R2_B04_DiffPressure_I						AT %I* 	:	UDINT;
	R2_B04_RemoteTemp2					AT %I* 	:	UDINT;
	R2_B04_HeatEnergyCounter_I				AT %I* 	:	UDINT;
	R2_B04_HeatDiffTemp						AT %I* 	:	UDINT;
	R2_B04_HeatPower						AT %I* 	:	UDINT;(* B0_SequenceNumber(1),B1AddressGenib(30),B2Class(11),B3Operation_Lenght(1),B4Data1(ID.34),Data(B5-B8) *)
	R2_B04_DirectDataReques_Temp_Geni		AT %Q* 	:	PB_GenibusType;
	R2_B04_DirectDataReply_Temp_Geni		AT %I* 	:	PB_GenibusType;

	R2_B04_NumberOfStarts					AT %I*	: 	UDINT;
	R2_B04_ActualSetpoint					AT %I*	:	UDINT;
	R2_B04_OperationTime					AT %I*	: 	UDINT;
	R2_B04_Speed							AT %I*	:	UDINT;
	R2_B04_Energy							AT %I*	: 	UDINT;
	R2_B04_Power							AT %I*	:	UDINT;
	R2_B04_PowerElectronicsTemp				AT %I*	:	UDINT;
	R2_B04_FaultCode						AT %I*	:	USINT;
	R2_B04_Volume							AT %I*	:	UDINT;
	R2_B04_WarningCode						AT %I*	:	USINT;


(*Gerät 6 (EL6731), BOX 05*)
(*DP/DP-Kopppler*)
(*DP_State*)
	R2_B05_PB_Zustand						AT %I*: USINT;
(*Daten*)
	R2_B05_StatusModule_I_Byte_1			AT %I*: USINT;
	R2_B05_StatusModule_I_Byte_2			AT %I*: USINT;
	R2_B05_StatusModule_I_Byte_5			AT %I*: USINT;
	R2_B05_StatusModule_I_Byte_6			AT %I*: USINT;
	R2_B05_ControlModule_O					AT %Q* :ARRAY [0..4] OF USINT;
	R2_B05_VolumeFlow_I						AT %I* :UDINT;
	R2_B05_PumpLiquidTemp_I					AT %I* :UDINT;
	R2_B05_OperationTime_I					AT %I* :UDINT;
	R2_B05_ActualSetpoint_I					AT %I* :UDINT;
	R2_B05_Frequency_I						AT %I* :UDINT;
	R2_B05_UserSetpoint_I					AT %I* :UDINT;
	R2_B05_DiffPressure_I					AT %I* :UDINT;
	R2_B05_RemoteTemp2						AT %I* :UDINT;
	R2_B05_HeatEnergyCounter_I				AT %I* :UDINT;
	R2_B05_HeatDiffTemp						AT %I* :UDINT;
	R2_B05_HeatPower						AT %I* :UDINT;(* B0_SequenceNumber(1),B1AddressGenib(30),B2Class(11),B3Operation_Lenght(1),B4Data1(ID.34),Data(B5-B8) *)
	R2_B05_DirectDataReques_Temp_Geni		AT %Q* :PB_GenibusType;
	R2_B05_DirectDataReply_Temp_Geni		AT %I* :PB_GenibusType;

	R2_B05_NumberOfStarts					AT %I*	: 	UDINT;
	R2_B05_ActualSetpoint					AT %I*	:	UDINT;
	R2_B05_OperationTime					AT %I*	: 	UDINT;
	R2_B05_Speed							AT %I*	:	UDINT;
	R2_B05_Energy							AT %I*	: 	UDINT;
	R2_B05_Power							AT %I*	:	UDINT;
	R2_B05_PowerElectronicsTemp				AT %I*	:	UDINT;
	R2_B05_FaultCode						AT %I*	:	USINT;
	R2_B05_Volume							AT %I*	:	UDINT;
	R2_B05_WarningCode						AT %I*	:	USINT;


(*Gerät 6 (EL6731), BOX 06*)
(*DP/DP-Kopppler*)
(*DP_State*)
	R2_B06_PB_Zustand						AT %I*: USINT;
(*Daten*)
	R2_B06_StatusModule_I_Byte_1			AT %I*: USINT;
	R2_B06_StatusModule_I_Byte_2			AT %I*: USINT;
	R2_B06_StatusModule_I_Byte_5			AT %I*: USINT;
	R2_B06_StatusModule_I_Byte_6			AT %I*: USINT;
	R2_B06_ControlModule_O					AT %Q* :ARRAY [0..4] OF USINT;
	R2_B06_VolumeFlow_I						AT %I* :UDINT;
	R2_B06_PumpLiquidTemp_I					AT %I* :UDINT;
	R2_B06_OperationTime_I					AT %I* :UDINT;
	R2_B06_ActualSetpoint_I					AT %I* :UDINT;
	R2_B06_Frequency_I						AT %I* :UDINT;
	R2_B06_UserSetpoint_I					AT %I* :UDINT;
	R2_B06_DiffPressure_I					AT %I* :UDINT;
	R2_B06_RemoteTemp2						AT %I* :UDINT;
	R2_B06_HeatEnergyCounter_I				AT %I* :UDINT;
	R2_B06_HeatDiffTemp						AT %I* :UDINT;
	R2_B06_HeatPower						AT %I* :UDINT;(* B0_SequenceNumber(1),B1AddressGenib(30),B2Class(11),B3Operation_Lenght(1),B4Data1(ID.34),Data(B5-B8) *)
	R2_B06_DirectDataReques_Temp_Geni		AT %Q* :PB_GenibusType;
	R2_B06_DirectDataReply_Temp_Geni		AT %I* :PB_GenibusType;

	R2_B06_NumberOfStarts					AT %I*	: 	UDINT;
	R2_B06_ActualSetpoint					AT %I*	:	UDINT;
	R2_B06_OperationTime					AT %I*	: 	UDINT;
	R2_B06_Speed							AT %I*	:	UDINT;
	R2_B06_Energy							AT %I*	: 	UDINT;
	R2_B06_Power							AT %I*	:	UDINT;
	R2_B06_PowerElectronicsTemp				AT %I*	:	UDINT;
	R2_B06_FaultCode						AT %I*	:	USINT;
	R2_B06_Volume							AT %I*	:	UDINT;
	R2_B06_WarningCode						AT %I*	:	USINT;

*)

END_VAR

(* stored: Version 1.1.0.1, ProductVersion 3.1.4024.9
   GVL Profibus: Id {6c6b23d2-5958-4ce2-aaec-fa070f52f6cf} *)
